SUBAPPLICATION TOGGLE_RPC_MASTER_QXA_OPC (* Klick-Toggle-'Kopf' fuer eine Gruppe von bis zu 6 gleichzeitig geschalteten Kanaelen OHNE eigenen physischen Ausgang: RPC-Trigger (CREATE_METHOD/SERVER_0) taktet ein AX_T_FF, dessen Zustand ueber 6 AX-Plugs (OUT1..OUT6) an Geschwister-SubApps (je ein AX_TON_MERGE_QXA_OPC pro Kanal) weitergereicht wird UND lokal publiziert wird, damit das Bedienmodul den Zustand als Hintergrundfarbe zeigen kann. Ungenutzte OUTn-Plugs bleiben einfach unverdrahtet. Fuer EINEN Ausgang stattdessen TOGGLE_RPC_MERGE_QXA_OPC verwenden (hat den physischen Ausgang schon eingebaut). *)
  (* Standard: 61499-2; Description: Copyright (c) 2026 Meisterschulen am Ostbahnhof This program and the accompanying materials are made available under the terms of the Eclipse Public License 2.0 which is available at https://www.eclipse.org/legal/epl-2.0/ SPDX-License-Identifier: EPL-2.0 *)
  (* Version 1.2, 2026-09-09, Franz Höpfinger, Meisterschulen am Ostbahnhof, Fix: TRIGGER_SERVER.RSP war nie verdrahtet - blockierte den OPC-UA-Server-Thread bis zu 4s (haelt open62541s globalen serviceMutex), verzoegerte dadurch JEDE OPC-UA-Statusmeldung projektweit. IND->RSP direkt verdrahtet. Siehe OPC_UA_VERNETZUNG.md Punkt 12. *)
  (* Version 1.1, 2026-09-07, Franz Höpfinger, Meisterschulen am Ostbahnhof, OUT-Plug durch OUT1..OUT6 (AX_SPLIT_7 statt AX_SPLIT_2) ersetzt - Adapter-Verbindungen sind 1:1, ein einzelner Plug kann nicht an mehrere Sockets gleichzeitig verdrahtet werden *)
  (* Version 1.0, 2026-09-07, Franz Höpfinger, Meisterschulen am Ostbahnhof, initial API and implementation and/or initial documentation - fuer Scheinwerfer (6 Kanaele, 1 SoftKey, versetztes Einschalten gegen kapazitive Einschaltstrom-Spitzen) *)
  PACKAGE MyLib::sys;
  (* Documentation:
  Klick-Toggle-Kopf ohne eigenen Ausgang (fuer Kanalgruppen bis 6)
   Wie Softkey_Toggle_RPC_TO_Remote_BG_OPC/Toggle_RPC_FROM_Remote_QXA_OPC, aber ohne physischen Ausgang - stattdessen wird der Toggle-Zustand ueber 6 eigene OUTn-Plugs an bis zu 6 Geschwister-SubApps im selben Netzwerk weitergegeben (z.B. mehrere AX_TON_MERGE_QXA_OPC-Instanzen, je eine pro physischem Kanal - Adapter-Verbindungen sind 1:1, deshalb kein einzelner gemeinsamer Plug fuer alle Kanaele). So kann EIN SoftKey mehrere Ausgaenge gleichzeitig toggeln, jeder Kanal aber trotzdem individuell zeitversetzt hochfahren (siehe AX_TON_MERGE_QXA_OPC.PT) - z.B. Scheinwerfer-Bank gegen kapazitive Einschaltstrom-Spitzen. Werden weniger als 6 Kanaele gebraucht, bleiben die restlichen OUTn-Plugs einfach unverdrahtet.
  *)
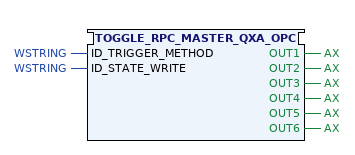
  VAR_INPUT
    ID_TRIGGER_METHOD : WSTRING; (* Lokale Methodenadresse (ACTION=CREATE_METHOD) fuer den argumentlosen Toggle-Trigger, wird vom Bedienmodul per CALL_METHOD aufgerufen *)
    ID_STATE_WRITE : WSTRING; (* Lokale Publish-Adresse (ACTION=WRITE) fuer den tatsaechlichen Toggle-Zustand - wird vom Bedienmodul remote abonniert (z.B. fuer GreenWhiteBackground) *)
  END_VAR
  PLUGS
    OUT1 : adapter::types::unidirectional::AX; (* Toggle-Zustand fuer Kanal 1 (z.B. AX_TON_MERGE_QXA_OPC.MASTER) *)
    OUT2 : adapter::types::unidirectional::AX; (* Toggle-Zustand fuer Kanal 2 *)
    OUT3 : adapter::types::unidirectional::AX; (* Toggle-Zustand fuer Kanal 3 *)
    OUT4 : adapter::types::unidirectional::AX; (* Toggle-Zustand fuer Kanal 4 *)
    OUT5 : adapter::types::unidirectional::AX; (* Toggle-Zustand fuer Kanal 5 *)
    OUT6 : adapter::types::unidirectional::AX; (* Toggle-Zustand fuer Kanal 6 *)
  END_PLUGS
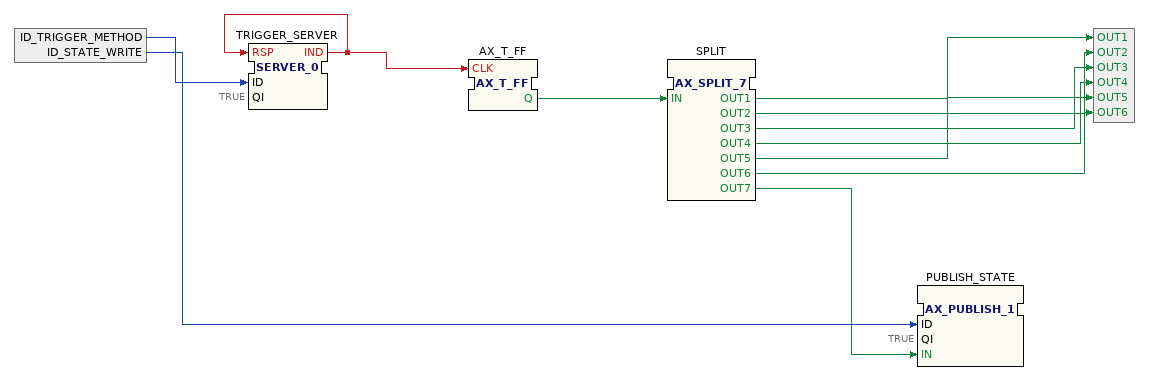
  FBS
    TRIGGER_SERVER : iec61499::net::SERVER_0(QI := TRUE);
    AX_T_FF : adapter::events::unidirectional::AX_T_FF;
    SPLIT : adapter::events::unidirectional::AX_SPLIT_7;
    PUBLISH_STATE : adapter::net::AX_PUBLISH_1(QI := TRUE);
  END_FBS
  EVENT_CONNECTIONS
    TRIGGER_SERVER.IND TO AX_T_FF.CLK;
    TRIGGER_SERVER.IND TO TRIGGER_SERVER.RSP;
  END_CONNECTIONS
  DATA_CONNECTIONS
    ID_TRIGGER_METHOD TO TRIGGER_SERVER.ID;
    ID_STATE_WRITE TO PUBLISH_STATE.ID;
  END_CONNECTIONS
  ADAPTER_CONNECTIONS
    AX_T_FF.Q TO SPLIT.IN;
    SPLIT.OUT1 TO OUT1;
    SPLIT.OUT2 TO OUT2;
    SPLIT.OUT3 TO OUT3;
    SPLIT.OUT4 TO OUT4;
    SPLIT.OUT5 TO OUT5;
    SPLIT.OUT6 TO OUT6;
    SPLIT.OUT7 TO PUBLISH_STATE.IN;
  END_CONNECTIONS
END_SUBAPPLICATION
